// TIA Portal V17 export
// export: Created 2026-04-13T11:12:04.3937976Z, ExportSetting WithDefaults, DisplayName Totally Integrated Automation Portal, DisplayVersion V17 Update 4, DisplayName TIA Portal Openness, DisplayVersion V17 Update 4, DisplayName TIA Portal Version Control Interface, DisplayVersion V17, DisplayName SINAMICS Startdrive Advanced, DisplayVersion V17, DisplayName SINAMICS Startdrive G130, G150, S120, S150, SINAMICS MV, S210, DisplayVersion V17, DisplayName SINAMICS Startdrive G110M, G120, G120C, G120D, G120P, G115D, DisplayVersion V17, DisplayName STEP 7 Professional, DisplayVersion V17 Update 4, DisplayName STEP 7 Safety, DisplayVersion V17, DisplayName WinCC Professional, DisplayVersion V17 Update 4
DATA_BLOCK "SV"   // DB14
{ S7_Optimized_Access := 'FALSE' }
VERSION : 0.1
// stored: AutoNumber true, DBAccessibleFromOPCUA true, DBAccessibleFromWebserver true, IsOnlyStoredInLoadMemory false, IsWriteProtectedInAS false
   VAR RETAIN
      BD布袋压差高报 : Real := 3000.0;
      BD布袋压差高高报 : Real := 3800.0;
      JF进风压差高报 : Real := 3000.0;
      JF进风压差高高报 : Real := 3800.0;
      TN塔内压力高高报 : Real := 14000.0;
      GD管道压力高报 : Real := 1500.0;
      GD管道压力高高报 : Real := 3000.0;
      GD管道压力设定 : Real := 700.0;
      TN塔内压力低报 : Real := -1000.0;
      TN塔内压力低低报 : Real := -1500.0;
      XH循风机频率设定 : Real := 35.0;
      YF引风频率设定 : Real := 30.0;
      JL进料泵频率设定 : Real := 11.0;
      JF进风温度设定 : Real := 110.0;
      CF出温异常设定 : Real := 0.0;
      JF进温高报 : Real := 220.0;
      JF进温高高报 : Real := 250.0;
      CF出风温度设定 : Real := 30.0;
      CF出温高报 : Real := 150.0;
      CF出温高高报 : Real := 200.0;
      WQ尾温高报 : Real := 35.0;
      WQ尾温高高报 : Real := 40.0;
      BD布袋反吹时间 : Real := 5.0;
      TW塔外气锤时间 : Real := 2.0;
      TN塔内气扫时间 : Real := 2.0;
      DQ氮气下限设定 : Real := 0.0;
      TN塔内压力高报 : Real := 11000.0;
      JW降温温度设定 : Real := 0.0;
      LS冷水温度写 : Real := 0.0;
      ZT主塔振打间隔 : Real := 0.0;
      TZ通针时间 : Real := 0.0;
      PM屏幕编号 : Real := 5.0;
      YH氧含仪高报 : Real := 5.0;
      JD进氮压力 : Real := 0.0;
      JL进料压力高报 : Real := 1500.0;
      JL进料压力高高报 : Real := 2000.0;
      WQ尾气温度 : Real := 35.0;
      JF进风保护温度 : Real := 50.0;
      YH氧含差值 : Real := 10.0;
      YH氧含仪1 : Real := 3.0;
      YH氧含仪2 : Real := 0.0;
      LS冷水检测写 : Real := 0.0;
      JF进风检测写 : Real := 0.0;
      QT气体检测仪低报 : Real := 0.0;
      QT气体检测仪低低报 : Real := 0.0;
      LX离心雾化 : Real := 42.0;
      DQ氮气加热写 : Real := 0.0;
      BD布袋振打时间 : Real := 0.0;
      PS排水延长时间 : Real := 0.0;
      AQ安全比例阀 : Real := 0.0;
      PK排空比例阀 : Real := 0.0;
      JB搅拌电机 : Real := 0.0;
      JF进风加热比例调节阀 : Real := 0.0;
      HF回风加热比例调节阀 : Real := 0.0;
      FK放空比例调节阀 : Real := 0.0;
      SF送风频率 : Real := 25.0;
      SS输送温度设定 : Real := 60.0;
      BD布袋出料设定 : Real := 0.0;
      YJ一级旋风出料设定 : Real := 0.0;
      EJ二级旋风出料设定 : Real := 0.0;
      BD布袋T出料设定 : Real := 0.0;
      YJ一级旋风T出料设定 : Real := 0.0;
      EJ二级旋风T出料设定 : Real := 0.0;
      BD布袋上阀开时间 : Real := 500.0;
      BD布袋上阀关时间 : Real := 3.0;
      BD布袋下阀开时间 : Real := 30.0;
      BD布袋下阀关时间 : Real := 3.0;
      YJ一级旋风上阀开时间 : Real := 300.0;
      YJ一级旋风上阀关时间 : Real := 3.0;
      YJ一级旋风下阀开时间 : Real := 30.0;
      YJ一级旋风下阀关时间 : Real := 3.0;
      EJ二级旋风上阀开时间 : Real := 400.0;
      EJ二级旋风上阀关时间 : Real := 3.0;
      EJ二级旋风下阀开时间 : Real := 30.0;
      EJ二级旋风下阀关时间 : Real := 3.0;
      HF回风温度设定 : Real := 0.0;
      ZT主塔压力设定 : Real := -200.0;
      KQ空气流量设定 : Real := 0.0;
      JL进料流量设定 : Real := 0.0;
      JL进料泵频率手动设定 : Real := 11.0;
      YF引风频率手动设定 : Real := 30.0;
      JF进风流量设定 : Real := 2400.0;
      YF引风频率自动设定 : Real := 30.0;
      JL进料频率自动设定 : Real := 11.0;
      FD阀导气压低报 : Real := 1.0;
      FD阀导气压低低报 : Real := 1.0;
      JF进风压差低报 : Real := 0.0;
      WH雾化油压低报 : Real := -1.0;
      WH雾化油压低低报 : Real := -1.0;
      JD进氮压力低报 : Real := 0.0;
      JD进氮压力低低报 : Real := 0.0;
      CF出风高效高报 : Real := 3000.0;
      CF出风高效高高报 : Real := 3800.0;
      CF出风高效低报 : Real := -50.0;
      SF输送高效高报 : Real := 0.0;
      SF输送高效高高报 : Real := 0.0;
      SF输送高效低报 : Real := 0.0;
      HF回风温度高报 : Real := 80.0;
      HF回风温度高高报 : Real := 100.0;
      BD布袋压差低报 : Real := -50.0;
      SS输送保护温度 : Real := 0.0;
      JL进料停机阈值 : Real := 30.0;
      SB设备振打间隔 : Real := 0.0;
      SS输送温度高高报 : Real := 110.0;
      SS输送温度高报 : Real := 102.0;
      SS输送压差高高报 : Real := 3800.0;
      SS输送压差高报 : Real := 3000.0;
      SS输送压差低报 : Real := -50.0;
      YJ一级液位高报 : Real := 400.0;
      YJ一级液位计高高报 : Real := 500.0;
      EJ二级液位计高报 : Real := 400.0;
      EJ二级液位计高高报 : Real := 500.0;
      CW除雾液位计高报 : Real := 400.0;
      CW除雾液位计高高报 : Real := 500.0;
      FD阀岛气压低报 : Real := 0.0;
      FD阀岛气压低低报 : Real := 0.0;
      YH氧含仪高高报 : Real := 12.0;
      JF进风流量低低报 : Real := 0.0;
      JF进风流量低报 : Real := 0.0;
      QZ前置水罐液位低报 : Real := 150.0;
      QZ前置水罐液位低低报 : Real := 100.0;
      JL进料流量低报 : Real := 0.0;
      JL进料流量低低报 : Real := 0.0;
      YJ一级旋风振打间隔 : Real := 6.0;
      EJ二级旋风振打间隔 : Real := 6.0;
      YJ一级旋风振荡运行 : Real := 3.0;
      YJ一级旋风振荡停止 : Real := 3.0;
      TJ调节单元 : Real := 4.0;
      TJ调节时间 : Real := 60.0;
      BD布袋压差自动反吹 : Real := 3500.0;
      BD布袋压差自动反吹时间 : Real := 1600.0;
      "ZT 中途停止温度分界" : Real := 115.0;
      JX碱洗温度设定 : Real := 0.0;
      FK放空阀手动设定 : Real := 0.0;
      FK放空阀自动设定 : Real := 0.0;
   END_VAR
BEGIN
END_DATA_BLOCK
